FUNCTION_BLOCK FB_Timer
VAR_INPUT
END_VAR
VAR_OUTPUT
	bDone			:BOOL;
	bBusy			:BOOL;
END_VAR
VAR
	_stateDelay			:INT;
	timerDelay			:TON;
END_VAR

METHOD Delay : BOOL
VAR_INPUT
	in			:TIME:=T#0S;	
END_VAR
VAR CONSTANT
	StateDone			:INT:=30;
END_VAR
CASE _stateDelay OF
	0:
		bDone := FALSE;
		timerDelay(IN:= FALSE);
		_stateDelay	:= 20;
	20:
		timerDelay(IN:=TRUE , PT:=in);
		IF timerDelay.Q THEN 
			bDone := TRUE;
			_stateDelay := StateDone;
		END_IF
END_CASE
END_METHOD

METHOD Reset : BOOL
VAR_INPUT
END_VAR
bDone := FALSE;

timerDelay(IN:=FALSE);

_stateDelay := 0;
END_METHOD

END_FUNCTION_BLOCK

(* stored: Version 1.1.0.1, ProductVersion 3.1.4022.16
   POU FB_Timer: Id {13b1ed0b-45cb-4272-a876-12621c72ae5b}, SpecialFunc None
   Method Delay: Id {134eed0e-cddb-4c30-bcbb-a8cb2bbaf357}
   Method Reset: Id {ef36a4a6-992e-4915-a31f-15de78a4d0af} *)
